   MachineConfig[14]."Unit Process"."EM - 340"."AV460-2".CW.ENABLE := True;
   MachineConfig[14]."Unit Dch"."EM - 222"."P222-1".CW.EXIST := False;
   MachineConfig[14]."Unit Dch"."EM - 222"."TS222-1".CW.ENABLE := true;
   MachineConfig[14]."Unit Dch"."EM - 300"."AV301-1".CW.ENABLE := True;
   MachineConfig[14]."Unit Dch"."EM - 300"."AV302-1".CW.ENABLE := True;
   MachineConfig[14]."Unit Dch"."EM - 300"."AV303-1".CW.ENABLE := True;
   MachineConfig[14]."Unit Dch"."EM - 300"."AV304-1".CW.ENABLE := True;
   MachineConfig[14]."Unit Dch"."EM - 300"."AV305-1".CW.ENABLE := True;
   MachineConfig[14]."Unit Dch"."EM - 300"."AV320-1".CW.ENABLE := True;
   MachineConfig[14]."Unit Dch"."EM - 300"."AV635-1".CW.ENABLE := True;
   MachineConfig[14]."Unit Dch"."EM - 375"."AV37X-1".CW.ENABLE := True;
   MachineConfig[14]."Unit Dch"."EM - 375"."PT37X-1".CW.ENABLE := True;
   MachineConfig[14]."Unit Dch"."EM - 375"."PT37X-1".CW.EXIST := False;
   MachineConfig[14]."Unit Dch"."EM - 506"."AV543-1".CW.ENABLE := True;
   MachineConfig[14]."Unit Dch"."EM - 506"."AV543-1".CW.EXIST := False;
   MachineConfig[14]."Unit Dch"."EM - 506".IP506a.CW.ENABLE := True;
   MachineConfig[14]."Unit Dch"."EM - 506"."PV376-1".CW.ENABLE := True;
   MachineConfig[14]."Unit Dch"."EM - 506"."PV376-1".CW.EXIST := False;
   MachineConfig[14]."Unit Dch"."EM - 506"."PV376-2".CW.ENABLE := True;
   MachineConfig[14]."Unit Dch"."EM - 506"."PV376-2".CW.EXIST := False;
   MachineConfig[14]."Unit Dch"."EM - 506".AVDCH.CW.ENABLE := true;

END_DATA_BLOCK

